(* IEC 61131-3 sources: ae-debugging/src/callpathExample, 3 files *)

(* ---- checks.st ---- *)
FUNCTION checkHundredth : BOOL
    VAR_INPUT
        count: int;
    END_VAR

    checkHundredth := (count MOD 100) = 0;
END_FUNCTION

(* ---- upcounter.st ---- *)
FUNCTION UpCounter_Func : Int
    VAR_INPUT
        up : Int;
    END_VAR

    VAR_TEMP
        up_temp : Int;
        down : Int;
    END_VAR

    up_temp := up + 1;
    down := up_temp - 2;
    UpCounter_Func := up_temp;
END_FUNCTION

FUNCTION Unused_Func : Bool
    ;
END_FUNCTION

(* ---- callpathExample.st ---- *)
PROGRAM UpCounter
    VAR_EXTERNAL
        CounterInt:       INT;
    END_VAR

    VAR_TEMP
        secondCounterIsEven: BOOL;
        isHundredth: BOOL;
    END_VAR

    CounterInt := UpCounter_Func(CounterInt);

    isHundredth := CheckHundredth(CounterInt);
    if isHundredth then
        CounterInt := UpCounter_Func(CounterInt);
    END_IF;

END_PROGRAM

PROGRAM SomeCounter
    VAR_EXTERNAL
        SecondCounterInt : Int;
    END_VAR

    SecondCounterInt := UpCounter_Func(SecondCounterInt);
END_PROGRAM
